TYPE PLCStruct :
STRUCT
    intVal		AT	%MB0	: 	INT;
    dintVal		AT	%MB2	: 	DINT;
    sintVal		AT	%MB6	: 	SINT;
    lrealVal	AT	%MB7	: 	LREAL;
    realVal		AT	%MB15	: 	REAL;
END_STRUCT
END_TYPE

(* stored: Version 1.1.0.1, ProductVersion 3.1.4024.10
   DUT PLCStruct: Id {27efefda-4b26-4341-b6ba-8f7451c0f3cb} *)
